PROGRAM MotorControlProgram
VAR
	rtCM_Start: R_TRIG;
	rtVM_Start: R_TRIG;
	rsCM	:	RS;
	rsVM	:	RS;
	
	targSpeed	:	INT;
END_VAR

(*
VAR_INPUT
	Run			:	BOOL;
	Direction	:	BOOL;
	ConstSpeed	:	BOOL;
	Velocity	:	INT;
END_VAR
VAR_OUTPUT
	isRunning	:	BOOL;
	iActualVel	:	INT;
END_VAR
*)



(* On / Off  Motor  *)

//***
rtCM_Start(CLK := GUI.bCMotor_Start);
rsCM(SET := rtCM_Start.Q);

Hardware.Motor2_Start := rsCM.Q1 ;


(*  TAMU  Motor  *)
//***
//rsVM(SET := GUI.bVMotor_Start);
//Hardware.Motor1_Start := rsVM.Q1 ;
Hardware.Motor1_Start :=  GUI.bVMotor_Start;
GUI.bVMotor_Running := Hardware.Motor1_Run_TAMU;
Hardware.Motor1_Constant_speed := GUI.bVMotor_ConstantSpeed;

// Y = x0 + %% * Xrng
targSpeed := REAL_TO_INT( 32767 * (GUI.iVMotor_TargetSpeed / 100.0) );
Hardware.Motor1_speed_value := targSpeed;

GUI.iVMotor_CurrentSpeed := REAL_TO_INT( Hardware.Motor1_real_value / 32767.0 * 100.0 );

END_PROGRAM

(* stored: Version 1.1.0.1, ProductVersion 3.1.4024.11
   POU MotorControlProgram: Id {00379d9c-0616-4665-8241-0c1fd684cd8f}, SpecialFunc None *)
